(* CoDeSys 2.3.9.47 project: ATS_P7_edgedetect.pro *)
(* Libraries: STANDARD.LIB 5.6.98 12:03:02 *)

(* Task configuration *)
TASK Standard (PRIORITY := 0, INTERVAL := T#10ms);
	MAIN
END_TASK

(* Global variable list: Global_Variables *)
VAR_GLOBAL
	(*Input Variables*)
	btnY	AT%I*	:BOOL; (*Button 1*)
	btnB	AT%I*	:BOOL; (*Button 2*)
	(*Output Variables*)
	lmpR	AT%Q*	:BOOL; (*Lamp 1*)
	lmpG	AT%Q*	:BOOL; (*Lamp 2*)
END_VAR

(* Global variable list: TwinCAT_Configuration *)
(* Generated automatically by TwinCAT - (read only) *)
VAR_CONFIG
	.btnY AT %IX0.0 : BOOL;	(*  ~ {LinkedWith:TIID^Device 1 (EtherCAT)^Term 1 (EK1200)^Term 2 (EL1004)^Channel 1^Input} *)
	.btnB AT %IX0.1 : BOOL;	(*  ~ {LinkedWith:TIID^Device 1 (EtherCAT)^Term 1 (EK1200)^Term 2 (EL1004)^Channel 2^Input} *)
	.lmpR AT %QX0.0 : BOOL;	(*  ~ {LinkedWith:TIID^Device 1 (EtherCAT)^Term 1 (EK1200)^Term 3 (EL2004)^Channel 1^Output} *)
	.lmpG AT %QX0.1 : BOOL;	(*  ~ {LinkedWith:TIID^Device 1 (EtherCAT)^Term 1 (EK1200)^Term 3 (EL2004)^Channel 2^Output} *)
END_VAR

(* Data type *)
TYPE T_STATE :
(
	STATE_IDLE := 0,
	STATE_RISE1:= 1,
	STATE_RISE2:= 2,
	STATE_FALL1:= 3,
	STATE_FALL2:= 4
);
END_TYPE

(* POU MAIN, ST *)
PROGRAM MAIN
VAR
	v_edgeDetect	: EdgeDetector;
	v_DedgeDetect	: DoubleEdgeDetector;
	isRising		: BOOL := FALSE;
	isFalling		: BOOL := FALSE;
	t				: REAL := 0;	(*Seconds*)
	tot				: REAL := 1;
END_VAR
(*Initialize*)
v_DedgeDetect();

(*Scan Button*)
v_DedgeDetect.sig_in 	:= btnY;
v_DedgeDetect.Ti 		:= tot;
v_DedgeDetect.t 		:= t;

(*Read Edge*)
IF v_DedgeDetect.rise = TRUE THEN
	lmpG := FALSE;
	lmpR := TRUE;
ELSIF v_DedgeDetect.rises = TRUE THEN
	lmpG := TRUE;
	lmpR := FALSE;
ELSE
	lmpG := FALSE;
	lmpR := FALSE;
END_IF

(*Show Edges*
lmpR		:= isFalling;
lmpG		:= isRising;
*)

(*Increment Time t*)
IF v_DedgeDetect.timer_ON = TRUE THEN
	(*Timer Starts counting*)
	t := t+0.01;
ELSE
	(*Used after Time is up*)
	t := 0;
END_IF
END_PROGRAM

(* POU EdgeDetector, ST *)
FUNCTION_BLOCK EdgeDetector
VAR_INPUT
	(*Input Signal*)
	sig_in 		: BOOL ;
END_VAR
VAR_OUTPUT
	(*Output Flags*)
	fall		: BOOL ;
	rise		: BOOL ;
END_VAR
VAR
	(*Lifelong Variables*)
	prev	: BOOL := FALSE;
END_VAR
IF (prev = sig_in) THEN
	(*NIL*)
	;
ELSIF (prev = TRUE) AND (sig_in = FALSE) THEN
	(*Falling Edge*)
	fall := TRUE;
	rise := FALSE;
ELSIF (prev = FALSE) AND (sig_in = TRUE) THEN
	(*Rising Edge*)
	fall := FALSE;
	rise := TRUE;
END_IF

(*Set current State = previous State*)
prev := sig_in;
END_FUNCTION_BLOCK

(* POU DoubleEdgeDetector, ST *)
FUNCTION_BLOCK DoubleEdgeDetector
VAR_INPUT
	(*Input Signal*)
	sig_in 		: BOOL ;
	(*Timer Count*)
	t			: REAL ;
	(*Idle Time*)
	Ti			: REAL ;
END_VAR
VAR_OUTPUT
	fall		: BOOL ;
	falls		: BOOL ;	
	rise		: BOOL ;
	rises		: BOOL ;
	(*Timer Commands*)
	timer_ON	: BOOL ;
END_VAR
VAR
	c_state		: T_STATE := STATE_IDLE;
	prev_sig	: BOOL := FALSE;
	edgeRise	: BOOL := FALSE;
	edgeFall	: BOOL := FALSE;
	TOF			: BOOL := FALSE;
END_VAR
(*Reset Outputs*)
DoubleEdgeDetector.fall		:= FALSE ;
DoubleEdgeDetector.falls	:= FALSE ;	
DoubleEdgeDetector.rise		:= FALSE ;
DoubleEdgeDetector.rises	:= FALSE ;

(*Check Timer Overflow*)
IF (t > Ti) THEN
	TOF := TRUE;
ELSE
	TOF := FALSE;
END_IF

(*Check Edge*)
IF (prev_sig = sig_in) THEN
	(*NIL*)
	edgeRise	:= FALSE;
	edgeFall	:= FALSE;
	;
ELSIF (prev_sig = TRUE) AND (sig_in = FALSE) THEN
	(*Falling Edge*)
	edgeFall := TRUE;
	edgeRise := FALSE;
ELSIF (prev_sig = FALSE) AND (sig_in = TRUE) THEN
	(*Rising Edge*)
	edgeFall := FALSE;
	edgeRise := TRUE;
END_IF

(*Set current Signal = previous Signal*)
prev_sig := sig_in;

(*Final State Machine Implementation*)
CASE c_state OF
	STATE_IDLE:
		(**)
		IF edgeRise = TRUE THEN
			c_state := STATE_RISE1;
		ELSIF edgeFall = TRUE THEN
			c_state := STATE_FALL1;
		ELSE
			c_state := STATE_IDLE;
		END_IF

	STATE_RISE1:
		(*Start Timer*)
		DoubleEdgeDetector.timer_ON := TRUE;
		(**)
		IF TOF = TRUE THEN
			DoubleEdgeDetector.timer_ON := FALSE;
			DoubleEdgeDetector.rise 	:= TRUE;
			c_state := STATE_IDLE;
		ELSIF edgeRise THEN 
			c_state := STATE_RISE2;
		ELSE
			c_state := STATE_RISE1;
		END_IF

	STATE_RISE2:
		(**)
		DoubleEdgeDetector.rises 	:= TRUE;
		c_state := STATE_IDLE;
		
	STATE_FALL1:
		(*Start Timer*)
		DoubleEdgeDetector.timer_ON := TRUE;
		(**)
		IF TOF = TRUE THEN
			DoubleEdgeDetector.timer_ON := FALSE;
			DoubleEdgeDetector.fall 	:= TRUE;
			c_state := STATE_IDLE;
		ELSIF edgeFall THEN 
			c_state := STATE_FALL2;
		ELSE
			c_state := STATE_FALL1;
		END_IF

	STATE_FALL2:
		(**)
		DoubleEdgeDetector.falls 	:= TRUE;
		c_state := STATE_IDLE;

	ELSE
		c_state := STATE_IDLE;
END_CASE;
END_FUNCTION_BLOCK
